GLOBALCONSTANTS zaehlstand (* Anzahl aktuell laufender Motoren als SINT (0..6), fuer AnlagenSequenz_06.ZAEHLSTAND, s. KONZEPT_Anlagensequenz.md *)
  (* Standard: 61499-1; Description: Copyright (c) 2026 HR Agrartechnik GmbH This program and the accompanying materials are made available under the terms of the Eclipse Public License 2.0 which is available at https://www.eclipse.org/legal/epl-2.0/ SPDX-License-Identifier: EPL-2.0 *)
  (* Version 1.0, 2026-08-25, Franz Höpfinger, HR Agrartechnik GmbH *)
  PACKAGE logiBUS::utils::sequence::const;
  VAR_GLOBAL CONSTANT
    ZAEHLSTAND_0 : SINT := SINT#0; (* 0 Motoren laufen (S_AUS) *)
    ZAEHLSTAND_1 : SINT := SINT#1; (* 1 Motor laeuft *)
    ZAEHLSTAND_2 : SINT := SINT#2; (* 2 Motoren laufen *)
    ZAEHLSTAND_3 : SINT := SINT#3; (* 3 Motoren laufen *)
    ZAEHLSTAND_4 : SINT := SINT#4; (* 4 Motoren laufen *)
    ZAEHLSTAND_5 : SINT := SINT#5; (* 5 Motoren laufen *)
    ZAEHLSTAND_6 : SINT := SINT#6; (* 6 Motoren laufen (S_LAEUFT, alle) *)
  END_VAR
END_GLOBALCONSTANTS
